// Mitsubishi GX Developer project: パレット移載装置   PLC: Q02

PROGRAM ERR-CODE
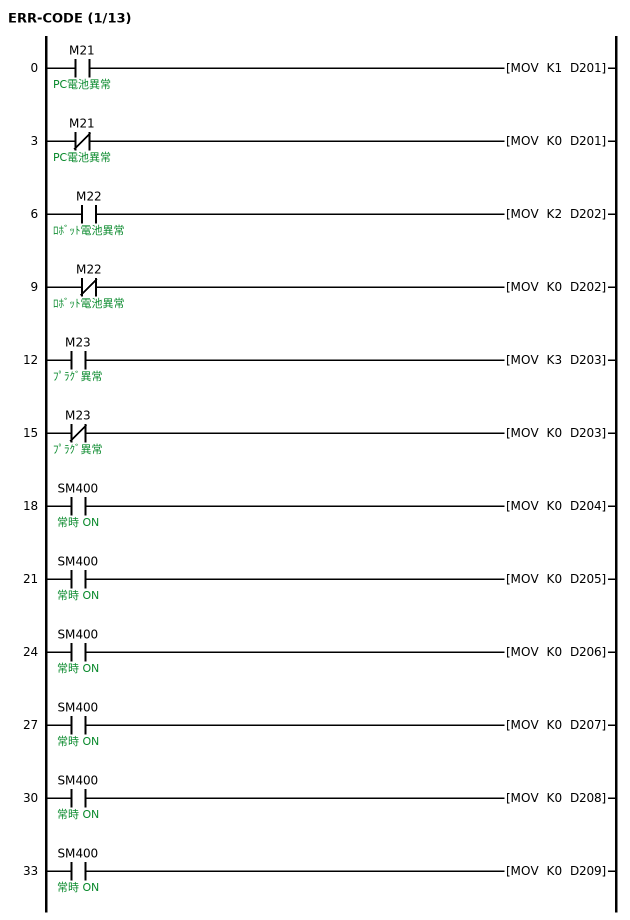
0     LD      M21  ; PC電池異常
      MOV     K1 D201
3     LDI     M21  ; PC電池異常
      MOV     K0 D201
6     LD      M22  ; ﾛﾎﾞｯﾄ電池異常
      MOV     K2 D202
9     LDI     M22  ; ﾛﾎﾞｯﾄ電池異常
      MOV     K0 D202
12    LD      M23  ; ﾌﾟﾗｸﾞ異常
      MOV     K3 D203
15    LDI     M23  ; ﾌﾟﾗｸﾞ異常
      MOV     K0 D203
18    LD      SM400  ; 常時 ON
      MOV     K0 D204
21    LD      SM400  ; 常時 ON
      MOV     K0 D205
24    LD      SM400  ; 常時 ON
      MOV     K0 D206
27    LD      SM400  ; 常時 ON
      MOV     K0 D207
30    LD      SM400  ; 常時 ON
      MOV     K0 D208
33    LD      SM400  ; 常時 ON
      MOV     K0 D209
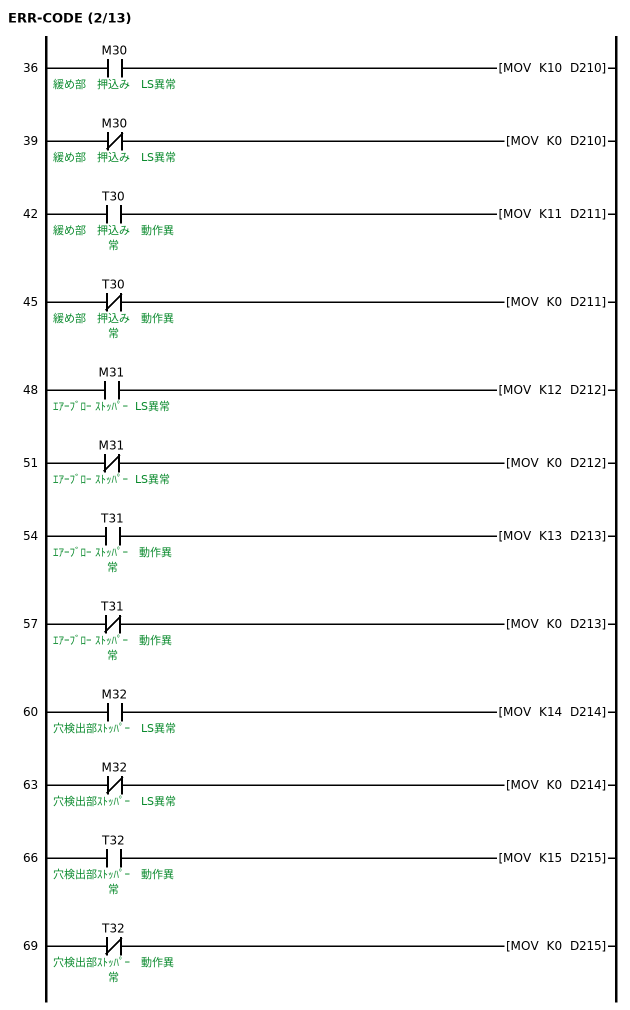
36    LD      M30  ; 緩め部　押込み　LS異常
      MOV     K10 D210
39    LDI     M30  ; 緩め部　押込み　LS異常
      MOV     K0 D210
42    LD      T30  ; 緩め部　押込み　動作異常
      MOV     K11 D211
45    LDI     T30  ; 緩め部　押込み　動作異常
      MOV     K0 D211
48    LD      M31  ; ｴｱｰﾌﾞﾛｰ ｽﾄｯﾊﾟｰ  LS異常
      MOV     K12 D212
51    LDI     M31  ; ｴｱｰﾌﾞﾛｰ ｽﾄｯﾊﾟｰ  LS異常
      MOV     K0 D212
54    LD      T31  ; ｴｱｰﾌﾞﾛｰ ｽﾄｯﾊﾟｰ　動作異常
      MOV     K13 D213
57    LDI     T31  ; ｴｱｰﾌﾞﾛｰ ｽﾄｯﾊﾟｰ　動作異常
      MOV     K0 D213
60    LD      M32  ; 穴検出部ｽﾄｯﾊﾟｰ　LS異常
      MOV     K14 D214
63    LDI     M32  ; 穴検出部ｽﾄｯﾊﾟｰ　LS異常
      MOV     K0 D214
66    LD      T32  ; 穴検出部ｽﾄｯﾊﾟｰ　動作異常
      MOV     K15 D215
69    LDI     T32  ; 穴検出部ｽﾄｯﾊﾟｰ　動作異常
      MOV     K0 D215
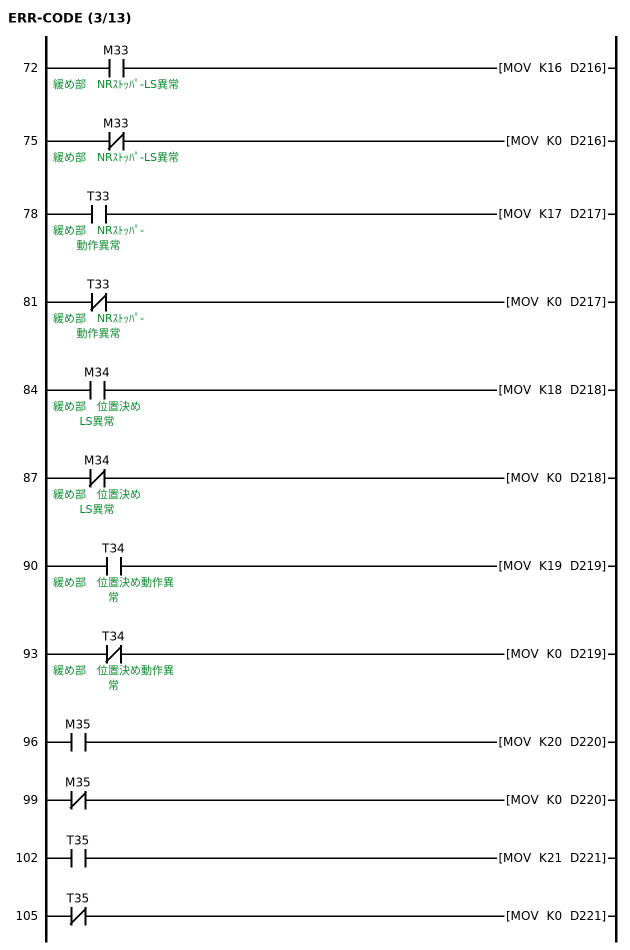
72    LD      M33  ; 緩め部　NRｽﾄｯﾊﾟ-LS異常
      MOV     K16 D216
75    LDI     M33  ; 緩め部　NRｽﾄｯﾊﾟ-LS異常
      MOV     K0 D216
78    LD      T33  ; 緩め部　NRｽﾄｯﾊﾟ-動作異常
      MOV     K17 D217
81    LDI     T33  ; 緩め部　NRｽﾄｯﾊﾟ-動作異常
      MOV     K0 D217
84    LD      M34  ; 緩め部　位置決め LS異常
      MOV     K18 D218
87    LDI     M34  ; 緩め部　位置決め LS異常
      MOV     K0 D218
90    LD      T34  ; 緩め部　位置決め動作異常
      MOV     K19 D219
93    LDI     T34  ; 緩め部　位置決め動作異常
      MOV     K0 D219
96    LD      M35
      MOV     K20 D220
99    LDI     M35
      MOV     K0 D220
102   LD      T35
      MOV     K21 D221
105   LDI     T35
      MOV     K0 D221
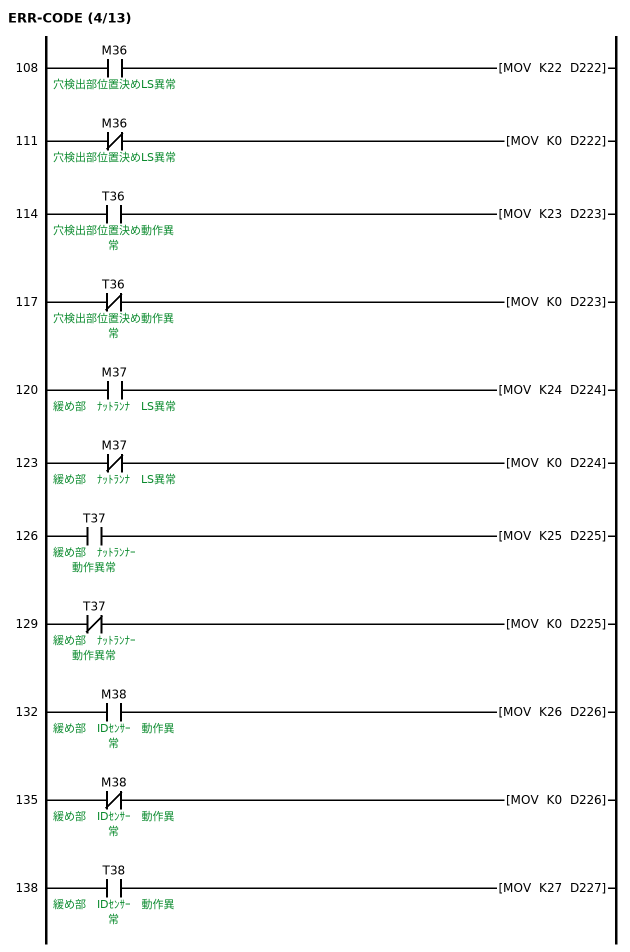
108   LD      M36  ; 穴検出部位置決めLS異常
      MOV     K22 D222
111   LDI     M36  ; 穴検出部位置決めLS異常
      MOV     K0 D222
114   LD      T36  ; 穴検出部位置決め動作異常
      MOV     K23 D223
117   LDI     T36  ; 穴検出部位置決め動作異常
      MOV     K0 D223
120   LD      M37  ; 緩め部　ﾅｯﾄﾗﾝﾅ　LS異常
      MOV     K24 D224
123   LDI     M37  ; 緩め部　ﾅｯﾄﾗﾝﾅ　LS異常
      MOV     K0 D224
126   LD      T37  ; 緩め部　ﾅｯﾄﾗﾝﾅｰ 動作異常
      MOV     K25 D225
129   LDI     T37  ; 緩め部　ﾅｯﾄﾗﾝﾅｰ 動作異常
      MOV     K0 D225
132   LD      M38  ; 緩め部　IDｾﾝｻｰ　動作異常
      MOV     K26 D226
135   LDI     M38  ; 緩め部　IDｾﾝｻｰ　動作異常
      MOV     K0 D226
138   LD      T38  ; 緩め部　IDｾﾝｻｰ　動作異常
      MOV     K27 D227
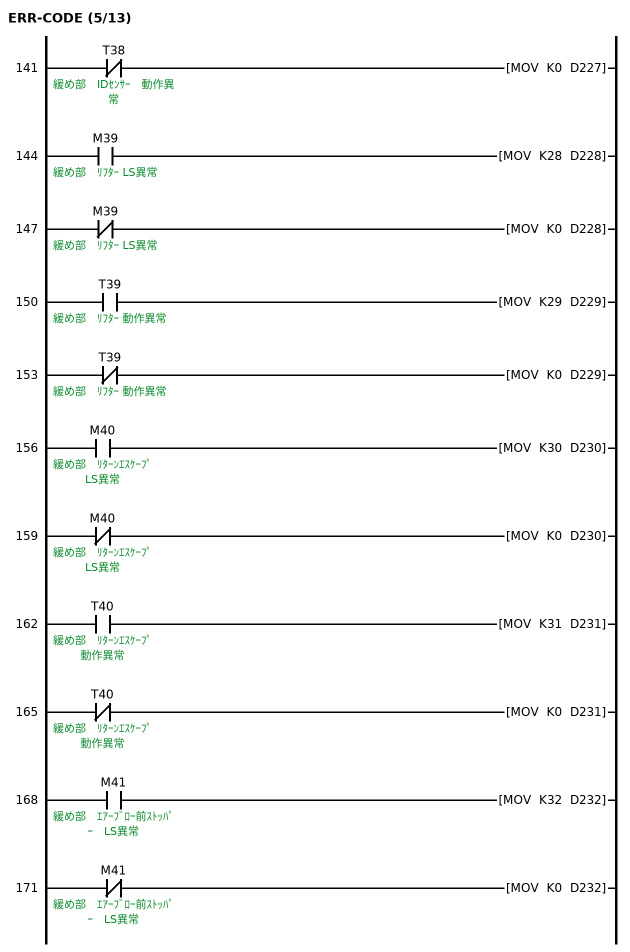
141   LDI     T38  ; 緩め部　IDｾﾝｻｰ　動作異常
      MOV     K0 D227
144   LD      M39  ; 緩め部　ﾘﾌﾀｰ LS異常
      MOV     K28 D228
147   LDI     M39  ; 緩め部　ﾘﾌﾀｰ LS異常
      MOV     K0 D228
150   LD      T39  ; 緩め部　ﾘﾌﾀｰ 動作異常
      MOV     K29 D229
153   LDI     T39  ; 緩め部　ﾘﾌﾀｰ 動作異常
      MOV     K0 D229
156   LD      M40  ; 緩め部　ﾘﾀｰﾝｴｽｹｰﾌﾟ LS異常
      MOV     K30 D230
159   LDI     M40  ; 緩め部　ﾘﾀｰﾝｴｽｹｰﾌﾟ LS異常
      MOV     K0 D230
162   LD      T40  ; 緩め部　ﾘﾀｰﾝｴｽｹｰﾌﾟ 動作異常
      MOV     K31 D231
165   LDI     T40  ; 緩め部　ﾘﾀｰﾝｴｽｹｰﾌﾟ 動作異常
      MOV     K0 D231
168   LD      M41  ; 緩め部　ｴｱｰﾌﾞﾛｰ前ｽﾄｯﾊﾟｰ　LS異常
      MOV     K32 D232
171   LDI     M41  ; 緩め部　ｴｱｰﾌﾞﾛｰ前ｽﾄｯﾊﾟｰ　LS異常
      MOV     K0 D232
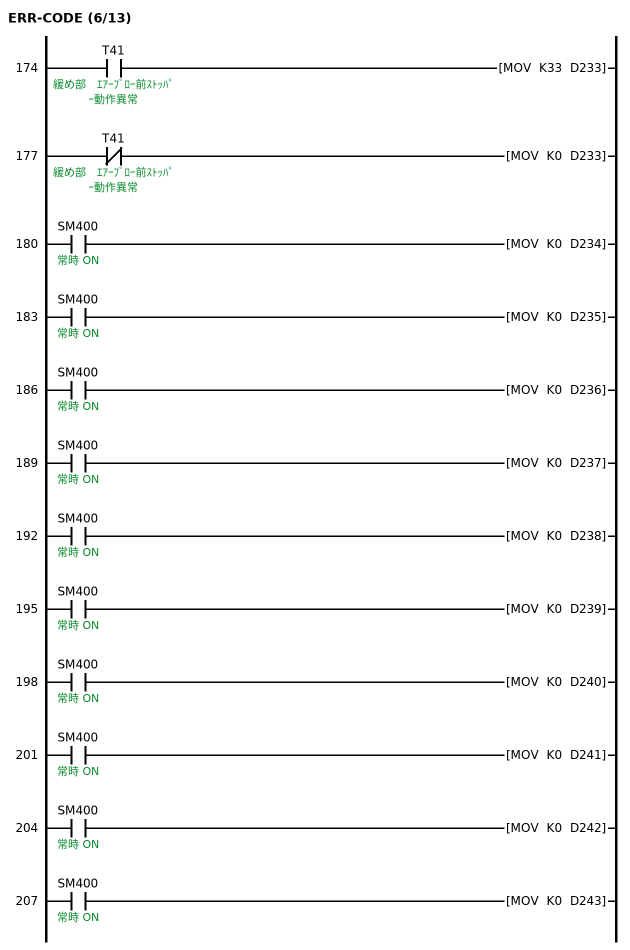
174   LD      T41  ; 緩め部　ｴｱｰﾌﾞﾛｰ前ｽﾄｯﾊﾟｰ動作異常
      MOV     K33 D233
177   LDI     T41  ; 緩め部　ｴｱｰﾌﾞﾛｰ前ｽﾄｯﾊﾟｰ動作異常
      MOV     K0 D233
180   LD      SM400  ; 常時 ON
      MOV     K0 D234
183   LD      SM400  ; 常時 ON
      MOV     K0 D235
186   LD      SM400  ; 常時 ON
      MOV     K0 D236
189   LD      SM400  ; 常時 ON
      MOV     K0 D237
192   LD      SM400  ; 常時 ON
      MOV     K0 D238
195   LD      SM400  ; 常時 ON
      MOV     K0 D239
198   LD      SM400  ; 常時 ON
      MOV     K0 D240
201   LD      SM400  ; 常時 ON
      MOV     K0 D241
204   LD      SM400  ; 常時 ON
      MOV     K0 D242
207   LD      SM400  ; 常時 ON
      MOV     K0 D243
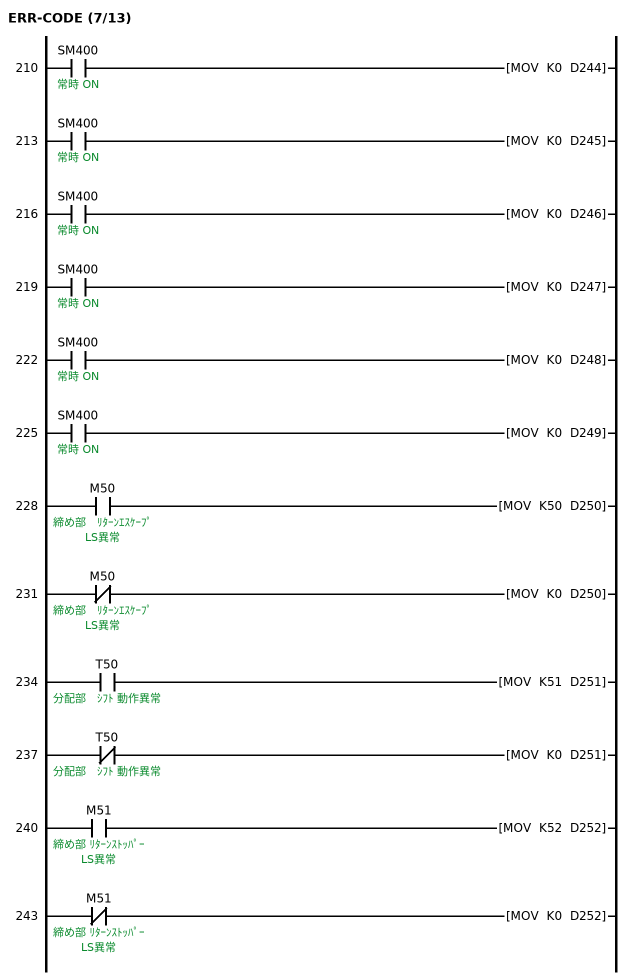
210   LD      SM400  ; 常時 ON
      MOV     K0 D244
213   LD      SM400  ; 常時 ON
      MOV     K0 D245
216   LD      SM400  ; 常時 ON
      MOV     K0 D246
219   LD      SM400  ; 常時 ON
      MOV     K0 D247
222   LD      SM400  ; 常時 ON
      MOV     K0 D248
225   LD      SM400  ; 常時 ON
      MOV     K0 D249
228   LD      M50  ; 締め部　ﾘﾀｰﾝｴｽｹｰﾌﾟ LS異常
      MOV     K50 D250
231   LDI     M50  ; 締め部　ﾘﾀｰﾝｴｽｹｰﾌﾟ LS異常
      MOV     K0 D250
234   LD      T50  ; 分配部　ｼﾌﾄ 動作異常
      MOV     K51 D251
237   LDI     T50  ; 分配部　ｼﾌﾄ 動作異常
      MOV     K0 D251
240   LD      M51  ; 締め部 ﾘﾀｰﾝｽﾄｯﾊﾟｰ LS異常
      MOV     K52 D252
243   LDI     M51  ; 締め部 ﾘﾀｰﾝｽﾄｯﾊﾟｰ LS異常
      MOV     K0 D252
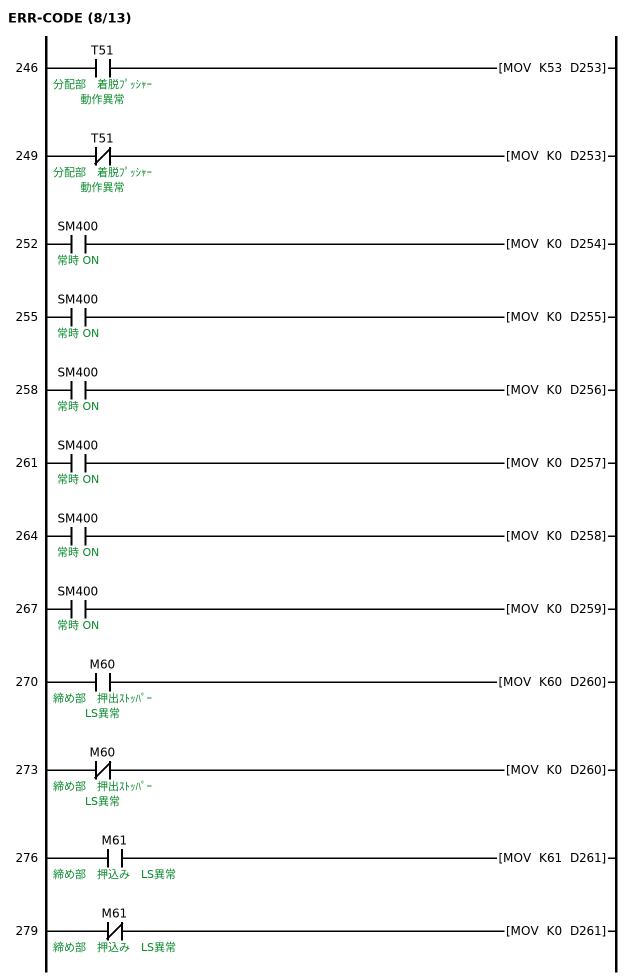
246   LD      T51  ; 分配部　着脱ﾌﾟｯｼｬｰ 動作異常
      MOV     K53 D253
249   LDI     T51  ; 分配部　着脱ﾌﾟｯｼｬｰ 動作異常
      MOV     K0 D253
252   LD      SM400  ; 常時 ON
      MOV     K0 D254
255   LD      SM400  ; 常時 ON
      MOV     K0 D255
258   LD      SM400  ; 常時 ON
      MOV     K0 D256
261   LD      SM400  ; 常時 ON
      MOV     K0 D257
264   LD      SM400  ; 常時 ON
      MOV     K0 D258
267   LD      SM400  ; 常時 ON
      MOV     K0 D259
270   LD      M60  ; 締め部　押出ｽﾄｯﾊﾟｰ LS異常
      MOV     K60 D260
273   LDI     M60  ; 締め部　押出ｽﾄｯﾊﾟｰ LS異常
      MOV     K0 D260
276   LD      M61  ; 締め部　押込み　LS異常
      MOV     K61 D261
279   LDI     M61  ; 締め部　押込み　LS異常
      MOV     K0 D261
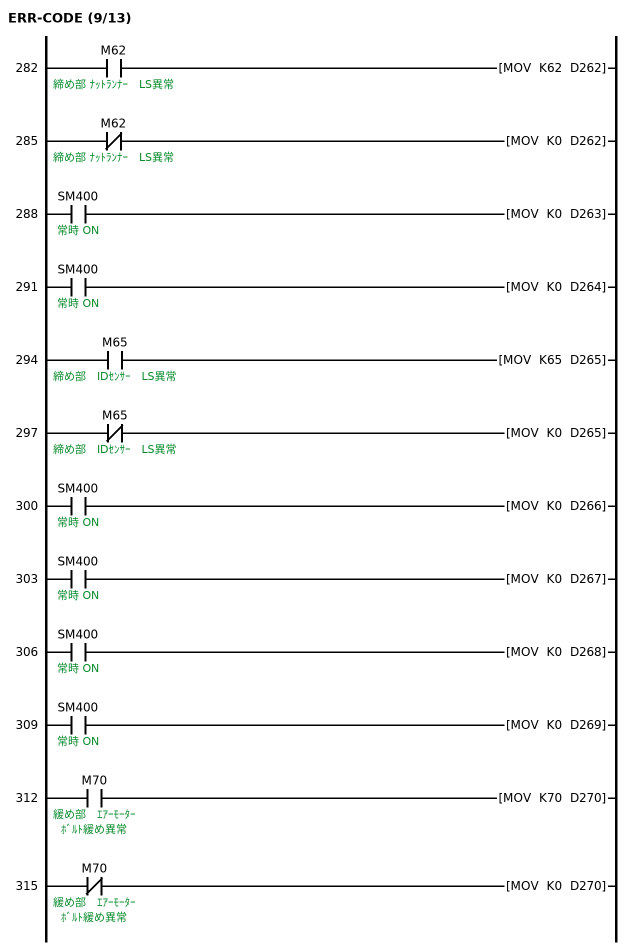
282   LD      M62  ; 締め部 ﾅｯﾄﾗﾝﾅｰ　LS異常
      MOV     K62 D262
285   LDI     M62  ; 締め部 ﾅｯﾄﾗﾝﾅｰ　LS異常
      MOV     K0 D262
288   LD      SM400  ; 常時 ON
      MOV     K0 D263
291   LD      SM400  ; 常時 ON
      MOV     K0 D264
294   LD      M65  ; 締め部　IDｾﾝｻｰ　LS異常
      MOV     K65 D265
297   LDI     M65  ; 締め部　IDｾﾝｻｰ　LS異常
      MOV     K0 D265
300   LD      SM400  ; 常時 ON
      MOV     K0 D266
303   LD      SM400  ; 常時 ON
      MOV     K0 D267
306   LD      SM400  ; 常時 ON
      MOV     K0 D268
309   LD      SM400  ; 常時 ON
      MOV     K0 D269
312   LD      M70  ; 緩め部　ｴｱｰﾓｰﾀｰ ﾎﾞﾙﾄ緩め異常
      MOV     K70 D270
315   LDI     M70  ; 緩め部　ｴｱｰﾓｰﾀｰ ﾎﾞﾙﾄ緩め異常
      MOV     K0 D270
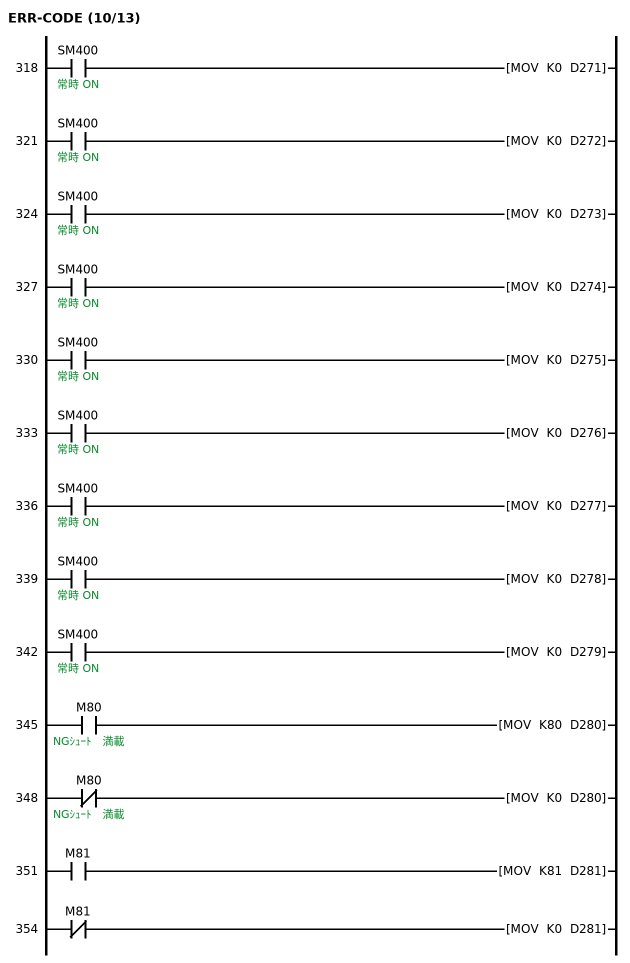
318   LD      SM400  ; 常時 ON
      MOV     K0 D271
321   LD      SM400  ; 常時 ON
      MOV     K0 D272
324   LD      SM400  ; 常時 ON
      MOV     K0 D273
327   LD      SM400  ; 常時 ON
      MOV     K0 D274
330   LD      SM400  ; 常時 ON
      MOV     K0 D275
333   LD      SM400  ; 常時 ON
      MOV     K0 D276
336   LD      SM400  ; 常時 ON
      MOV     K0 D277
339   LD      SM400  ; 常時 ON
      MOV     K0 D278
342   LD      SM400  ; 常時 ON
      MOV     K0 D279
345   LD      M80  ; NGｼｭｰﾄ　満載
      MOV     K80 D280
348   LDI     M80  ; NGｼｭｰﾄ　満載
      MOV     K0 D280
351   LD      M81
      MOV     K81 D281
354   LDI     M81
      MOV     K0 D281
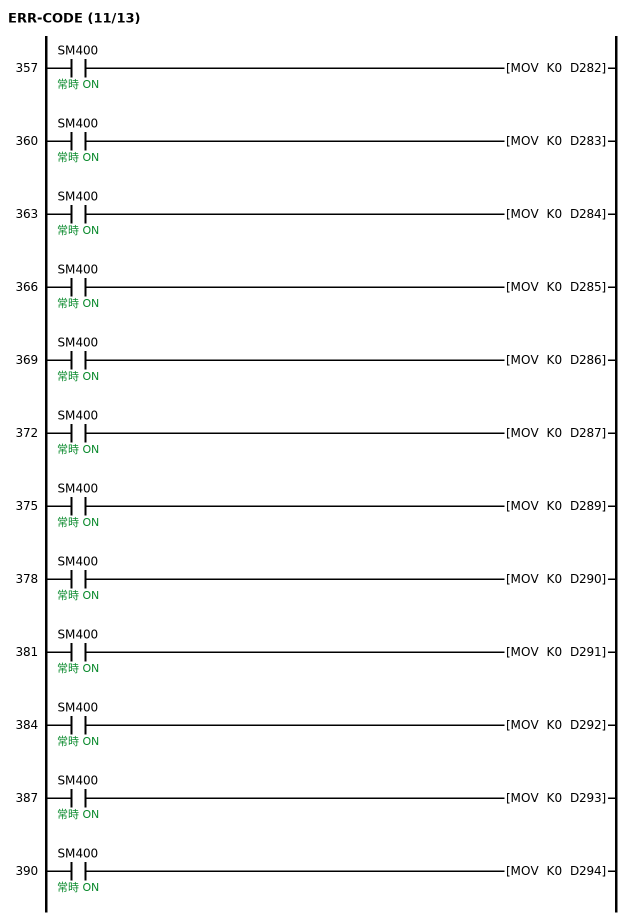
357   LD      SM400  ; 常時 ON
      MOV     K0 D282
360   LD      SM400  ; 常時 ON
      MOV     K0 D283
363   LD      SM400  ; 常時 ON
      MOV     K0 D284
366   LD      SM400  ; 常時 ON
      MOV     K0 D285
369   LD      SM400  ; 常時 ON
      MOV     K0 D286
372   LD      SM400  ; 常時 ON
      MOV     K0 D287
375   LD      SM400  ; 常時 ON
      MOV     K0 D289
378   LD      SM400  ; 常時 ON
      MOV     K0 D290
381   LD      SM400  ; 常時 ON
      MOV     K0 D291
384   LD      SM400  ; 常時 ON
      MOV     K0 D292
387   LD      SM400  ; 常時 ON
      MOV     K0 D293
390   LD      SM400  ; 常時 ON
      MOV     K0 D294
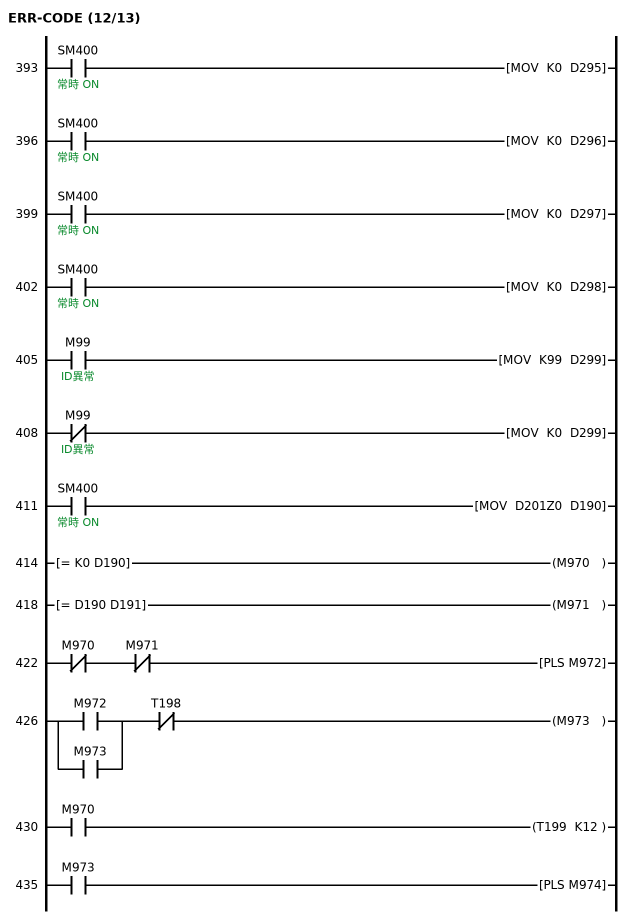
393   LD      SM400  ; 常時 ON
      MOV     K0 D295
396   LD      SM400  ; 常時 ON
      MOV     K0 D296
399   LD      SM400  ; 常時 ON
      MOV     K0 D297
402   LD      SM400  ; 常時 ON
      MOV     K0 D298
405   LD      M99  ; ID異常
      MOV     K99 D299
408   LDI     M99  ; ID異常
      MOV     K0 D299
411   LD      SM400  ; 常時 ON
      MOV     D201Z0 D190
414   LD=     K0 D190
      OUT     M970
418   LD=     D190 D191
      OUT     M971
422   LDI     M970
      ANI     M971
      PLS     M972
426   LD      M972
      OR      M973
      ANI     T198
      OUT     M973
430   LD      M970
      OUT     T199 K12
435   LD      M973
      PLS     M974
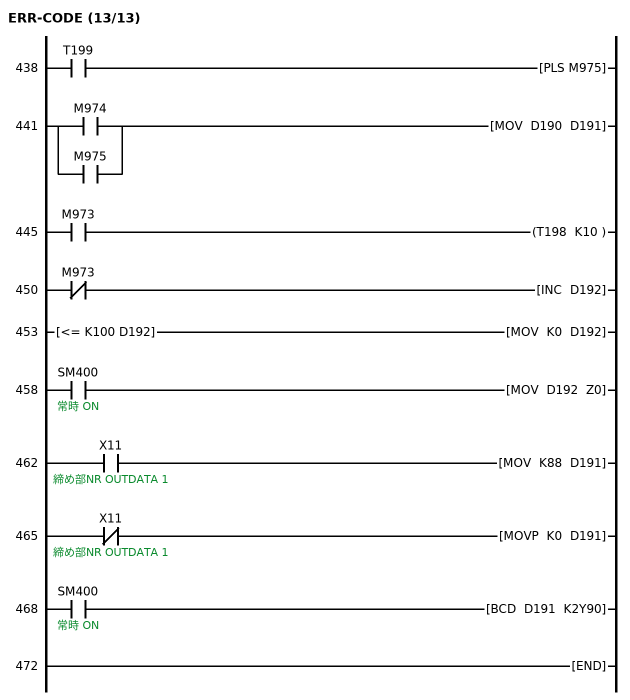
438   LD      T199
      PLS     M975
441   LD      M974
      OR      M975
      MOV     D190 D191
445   LD      M973
      OUT     T198 K10
450   LDI     M973
      INC     D192
453   LD<=    K100 D192
      MOV     K0 D192
458   LD      SM400  ; 常時 ON
      MOV     D192 Z0
462   LD      X11  ; 締め部NR OUTDATA 1
      MOV     K88 D191
465   LDI     X11  ; 締め部NR OUTDATA 1
      MOVP    K0 D191
468   LD      SM400  ; 常時 ON
      BCD     D191 K2Y90  ; 締め部NR　STOP
472   END
END_PROGRAM
